FUNCTION_BLOCK FB_DeviceWord EXTENDS FB_LinkDataWord
VAR_INPUT		
	nControl  			: BYTE;
	nControlData  		: WORD;
END_VAR

VAR_OUTPUT
	nStatus  			: BYTE;
	nStatusData  		: WORD;
END_VAR

SUPER^();
Control := nControl;
ControlData := nControlData;
nStatus := Status;
nStatusData := StatusData;

END_FUNCTION_BLOCK

(* stored: Version 1.1.0.1, ProductVersion 3.1.4024.12
   POU FB_DeviceWord: Id {58abdc43-a45f-0a4e-18ba-0ca1eadac5c7}, SpecialFunc None *)
